FUNCTION CheckOk : BOOL
VAR_INPUT
	hr : HRESULT;
END_VAR

CheckOk := (hr = S_OK);

END_FUNCTION

(* stored: Version 1.1.0.1, ProductVersion 3.1.4024.11
   POU CheckOk: Id {61f2d040-0588-4303-9eb6-4a66f7a53b42}, SpecialFunc None *)
